FUNCTION_BLOCK Std900FastAttenuation EXTENDS FastAttenuationBase
VAR_INPUT
END_VAR
VAR_OUTPUT
END_VAR
VAR
	{attribute 'OPC.UA.DA' := '0'}
	_config : Std900FastAttenuationConfig;
	{attribute 'OPC.UA.DA' := '0'}
	IoStd900 : IoStd900;
	
	{attribute 'OPC.UA.DA' := '0'}
	_deliverMessages : INT;
	
	PositionMsg : STRING(255);
	
	{region 'Commands'}	
		 
	{attribute 'OPC.UA.DA' := '0'}
	_moveAbsPosition	 : BOOL;
		 
	{endregion}
		 
	{attribute 'OPC.UA.DA' := '0'}
	_initDevice : BOOL;	
		
	{attribute 'OPC.UA.DA' := '0'}
	_pos : UINT;
	{attribute 'OPC.UA.DA' := '0'}
	_itemScheduler : INT;
	{attribute 'OPC.UA.DA' := '0'}
	_pulseGenerator : TON;		
END_VAR

// Init device
InitDevice(); 	
			  
// Deliver messages
CASE _deliverMessages OF	
		EFeedbackMsgStd900.PositionMsg :
		PositionMsg := REAL_TO_STRING(GetPosition());			
END_CASE
	
_deliverMessages := 0;

// Commands
MoveAbsPosition(_moveAbsPosition, _pos); 

IF NOT _moveAbsPosition THEN
	MessageScheduler();
END_IF

METHOD FB_init : BOOL
VAR_INPUT
	bInitRetains : BOOL; // if TRUE, the retain variables are initialized (warm start / cold start)
	bInCopyCode : BOOL;  // if TRUE, the instance afterwards gets moved into the copy code (online change)
	Config : Std900FastAttenuationConfig;
END_VAR
IF Config.IsEnabled THEN
	_config := Config;
	
	SUPER^._fastAttenuationConfig.Name := Config.Name;
	SUPER^._fastAttenuationConfig.DeviceID := Config.DeviceID;
	SUPER^._fastAttenuationConfig.IsEnabled := Config.IsEnabled;
	SUPER^._fastAttenuationConfig.LogLevel := Config.LogLevel;
	
	SUPER^.Name := Config.Name;
	SUPER^.DeviceID := Config.DeviceID;	
	THIS^.Family := DeviceFamily.FastAttenuation;
	
	_Logger.Information(_message.Reset().Append('Init ').
							Append('{').Append(TO_STRING(THIS^.Family)).Append('} - ').
							Append('{').Append(TO_STRING(Config.Name)).Append('}').ToString());																													
END_IF
END_METHOD

METHOD GetPosition : REAL
VAR_INPUT
END_VAR
_deliverMessages := EFeedbackMsgStd900.PositionMsg;

GetPosition := ((IoStd900.OutputPwm - Const.STD900_LOW_LIMIT) * Const.STD900_MAX_ANGLE) / (Const.STD900_HIGHT_LIMIT - Const.STD900_LOW_LIMIT);
END_METHOD

METHOD InitDevice : BOOL
VAR_INPUT
END_VAR
IF NOT _initDevice THEN	
	_logger.Information(_message.Reset().
								Append(_config.Name).
								Append(' - Init device').ToString());
							
	THIS^.Status := TExecutionState.Ready;
	
	IF IoStd900.OutputPwm = 0 THEN
		MoveAbsPosition(TRUE, 0);
	END_IF
	GetPosition();
	
	_initDevice := TRUE;	
END_IF
END_METHOD

METHOD MessageScheduler
VAR_INPUT
END_VAR
IF _pulseGenerator.Q THEN
	_pulseGenerator(IN := FALSE, PT := T#10MS);
		
	CASE _itemScheduler OF	
		0:	GetPosition();
			_itemScheduler := 1;	
		
		1 : 
			_itemScheduler := 0;											
	END_CASE
ELSE
	_pulseGenerator(IN := TRUE, PT := T#100MS);	
END_IF
END_METHOD

{attribute 'TcRpcEnable' := '1'}
METHOD PROTECTED MoveAbsPosition 
VAR_INPUT
	Execute : BOOL;
	AnglePosition : LREAL;
END_VAR
VAR
	pulseLength : LREAL;
END_VAR
IF Execute THEN
	_logger.Information(_message.Reset().
								Append(_config.Name).
								Append(' - Move absolute position : ').Append(TO_STRING(AnglePosition)).ToString());
	
	_moveAbsPosition := FALSE;
	
	IF AnglePosition >= Const.STD900_MIN_ANGLE AND AnglePosition <= Const.STD900_MAX_ANGLE THEN
		
		IF AnglePosition = Const.STD900_MIN_ANGLE THEN
			pulseLength := Const.STD900_LOW_LIMIT;		
		ELSE
			pulseLength := (Const.STD900_HIGHT_LIMIT - Const.STD900_LOW_LIMIT) / (Const.STD900_MAX_ANGLE / AnglePosition) + Const.STD900_LOW_LIMIT;
		END_IF
		
		_logger.Information(_message.Reset().
								Append('Pulse length : ').Append(TO_STRING(pulseLength)).
								Append(' µs').ToString());
		
		IoStd900.OutputPwm := LREAL_TO_UINT(pulseLength);
		IoStd900.OutputPeriodPwm := Const.STD900_INTERVAL + LREAL_TO_UINT(pulseLength);
	
	END_IF
	
	_itemScheduler := 0;
END_IF
END_METHOD

{attribute 'TcRpcEnable' := '1'}
METHOD RaisePropertiesChanged
VAR_INPUT
	Execute : BOOL;
END_VAR
IF Execute THEN
	PositionMsg := ' ';
END_IF
END_METHOD

END_FUNCTION_BLOCK

(* stored: Version 1.1.0.1, ProductVersion 3.1.4024.12
   POU Std900FastAttenuation: Id {a15326b2-c781-4242-993c-f6942d46b2cc}, SpecialFunc None
   Folder Commands: Id {6a7244d8-f986-48ab-8098-59846062eedd}
   Method FB_init: Id {70e7abd4-c246-4c8b-8cb5-0fd9b6f29999}
   Method GetPosition: Id {12ab734f-68bb-415f-ac8c-26f62606f20e}
   Method InitDevice: Id {b765d30f-351d-44d4-83de-9f71dc2f304c}
   Method MessageScheduler: Id {e123a467-c63b-4caf-b194-33f910ef3674}
   Method MoveAbsPosition: Id {abf85d58-59a8-4f6a-85f6-e0f76a6a9aea}
   Method RaisePropertiesChanged: Id {13543100-5dfa-4566-8a34-8a160d04283e} *)
